(*udt (user defined type) of Beckhoff EP6224-0002 - 4 Point IP67 Rated IO-Link Box:
	Version 20210621
		- initial creation, j.underhill

*)


TYPE udt_EP6224_I :
STRUCT
	Port1_I: BOOL;
	Port2_I: BOOL;
	Port3_I: BOOL;
	Port4_I: BOOL;

END_STRUCT
END_TYPE

(* stored: Version 1.1.0.1, ProductVersion 3.1.4024.9
   DUT udt_EP6224_I: Id {895fe964-1d10-455c-a7bf-d1a5fc51076b} *)
